// TIA Portal V19 export
ORGANIZATION_BLOCK "Main"   // OB1, LAD, ProgramCycle
TITLE = "Main Program Sweep (Cycle)"
{ S7_Optimized_Access := 'TRUE' }
// stored: SetENOAutomatically false
   VAR_INPUT
      Initial_Call : Bool;   // Initial call of this OB
      Remanence : Bool;   // =True, if remanent data are available
   END_VAR
   VAR_TEMP   // added for the SCL form of the ladder/FBD networks
      _w1 : Bool;
      _w2 : Bool;
      _w3 : Bool;
      _w4 : Bool;
      _w5 : Bool;
      _w6 : Bool;
      _w7 : Bool;
      _w8 : Bool;
      _w9 : Bool;
      _w10 : Bool;
   END_VAR
BEGIN

REGION Network 1: #SHIV
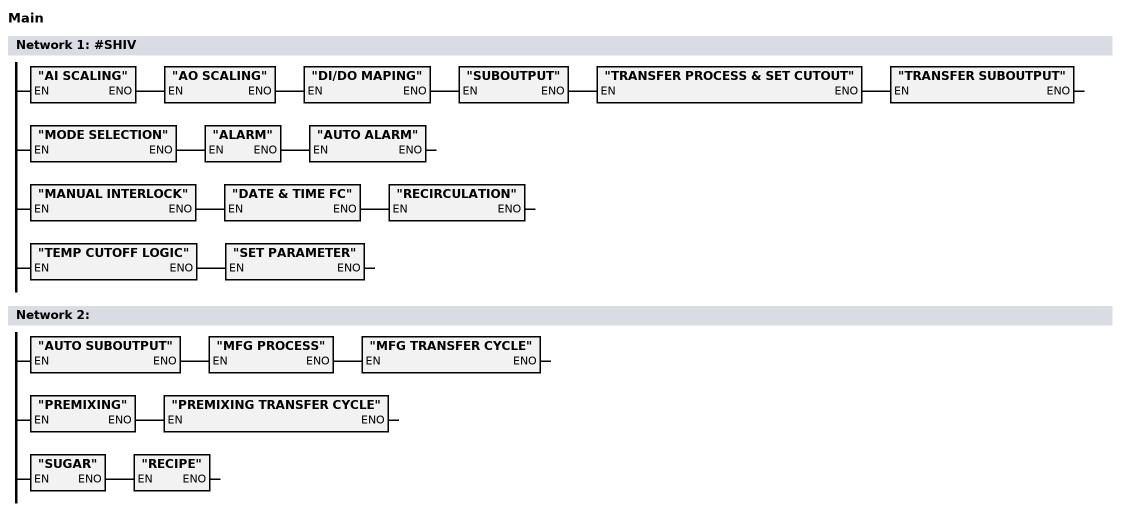
   RUNG wire#powerrail
      "AI SCALING"()
      "AO SCALING"()
      "DI/DO MAPING"()
      "SUBOUTPUT"()
      "TRANSFER PROCESS & SET CUTOUT"()
      "TRANSFER SUBOUTPUT"()
   END_RUNG
   RUNG wire#powerrail
      "MODE SELECTION"()
      "ALARM"()
      "AUTO ALARM"()
   END_RUNG
   RUNG wire#powerrail
      "MANUAL INTERLOCK"()
      "DATE & TIME FC"()
      "RECIRCULATION"()
   END_RUNG
   RUNG wire#powerrail
      "TEMP CUTOFF LOGIC"()
      "SET PARAMETER"()
   END_RUNG
   // the same network as SCL:
   "AI SCALING"(ENO => #_w1);
   "AO SCALING"(EN := #_w1, ENO => #_w2);
   "DI/DO MAPING"(EN := #_w2, ENO => #_w3);
   "SUBOUTPUT"(EN := #_w3, ENO => #_w4);
   "TRANSFER PROCESS & SET CUTOUT"(EN := #_w4, ENO => #_w5);
   IF #_w5 THEN "TRANSFER SUBOUTPUT"(); END_IF;
   "MODE SELECTION"(ENO => #_w6);
   "ALARM"(EN := #_w6, ENO => #_w7);
   IF #_w7 THEN "AUTO ALARM"(); END_IF;
   "MANUAL INTERLOCK"(ENO => #_w8);
   "DATE & TIME FC"(EN := #_w8, ENO => #_w9);
   IF #_w9 THEN "RECIRCULATION"(); END_IF;
   "TEMP CUTOFF LOGIC"(ENO => #_w10);
   IF #_w10 THEN "SET PARAMETER"(); END_IF;
END_REGION

REGION Network 2
   RUNG wire#powerrail
      "AUTO SUBOUTPUT"()
      "MFG PROCESS"()
      "MFG TRANSFER CYCLE"()
   END_RUNG
   RUNG wire#powerrail
      "PREMIXING"()
      "PREMIXING TRANSFER CYCLE"()
   END_RUNG
   RUNG wire#powerrail
      "SUGAR"()
      "RECIPE"()
   END_RUNG
   // the same network as SCL:
   "AUTO SUBOUTPUT"(ENO => #_w1);
   "MFG PROCESS"(EN := #_w1, ENO => #_w2);
   IF #_w2 THEN "MFG TRANSFER CYCLE"(); END_IF;
   "PREMIXING"(ENO => #_w3);
   IF #_w3 THEN "PREMIXING TRANSFER CYCLE"(); END_IF;
   "SUGAR"(ENO => #_w4);
   IF #_w4 THEN "RECIPE"(); END_IF;
END_REGION
END_ORGANIZATION_BLOCK
